(* Logix 5000 project; controller ARS14002_PLC vendor 1 type 14 code 218 rev 30.11; software revision 30.01; part 2 of 13 *)
(* tags used below, declared in another part *)
   FCV_1001 : CM_AO_VLV;
   FCV_1002 : CM_AO_VLV;
   FCV_101A : CM_AO_VLV;
   FCV_101B : CM_AO_VLV;
   FCV_101C : CM_AO_VLV;
   FCV_102A : CM_AO_VLV;
   FCV_102B : CM_AO_VLV;
   FCV_102C : CM_AO_VLV;
   FCV_1221 : CM_AO_VLV;
   FCV_1251 : CM_AO_VLV;
   FCV_202 : CM_AO_VLV;
   FCV_204 : CM_AO_VLV;
   FCV_207 : CM_AO_VLV;
   FCV_504 : CM_AO_VLV;
   FCV_603 : CM_AO_VLV;
   FCV_605 : CM_AO_VLV;
   FCV_753 : CM_AO_VLV;
   FCV_754 : CM_AO_VLV;
   FCV_755 : CM_AO_VLV;
   FT_1002 : CM_AI_SCL;
   FT_1002_MAVE : REAL;
   FT_1002_MAVE_STORAGE : REAL[30];
   FT_1221 : CM_AI_SCL;
   FT_1251 : CM_AI_SCL;
   PDT_603 : CM_AI_SCL_ALT;
   PDT_751 : CM_AI_SCL_ALT;
   PDT_753 : CM_AI_SCL_ALT;
   PT_1001 : CM_AI_SCL;
   PT_101A : CM_AI_SCL;
   PT_101B : CM_AI_SCL;
   PT_101C : CM_AI_SCL;
   PT_201 : CM_AI_SCL;
   PT_601 : CM_AI_SCL;
   PT_701 : CM_AI_SCL;
   PT_753 : CM_AI_SCL;
   PT_902 : CM_AI_SCL;
   SV_1001F : CM_DO_GENERIC;
   SV_1002F : CM_DO_GENERIC;
   SV_101AF : CM_DO_GENERIC;
   SV_101BF : CM_DO_GENERIC;
   SV_101CF : CM_DO_GENERIC;
   SV_102AF : CM_DO_GENERIC;
   SV_102BF : CM_DO_GENERIC;
   SV_102CF : CM_DO_GENERIC;
   SV_1221F : CM_DO_GENERIC;
   SV_1251F : CM_DO_GENERIC;
   SV_202F : CM_DO_GENERIC;
   SV_204F : CM_DO_GENERIC;
   SV_207F : CM_DO_GENERIC;
   SV_504F : CM_DO_GENERIC;
   SV_603F : CM_DO_GENERIC;
   SV_605F : CM_DO_GENERIC;
   SV_753F : CM_DO_GENERIC;
   SV_754F : CM_DO_GENERIC;
   SV_755F : CM_DO_GENERIC;

   TE_1250A : CM_AI_SCL := (RawMin := -4500, RawMax := 10000, EuMin := -450.0, EuMax := 1000.0, In_Raw := 487, Percent := 4.8700013, PV := 48.700012);
   TE_1250B : CM_AI_SCL := (RawMin := -4500, RawMax := 10000, EuMin := -450.0, EuMax := 1000.0, In_Raw := 520, Percent := 5.2000003, PV := 52.0);
   TE_1252 : CM_AI_SCL := (RawMin := -4500, RawMax := 10000, EuMin := -450.0, EuMax := 1000.0, In_Raw := 528, Percent := 5.279999, PV := 52.799988);
   TE_501 : CM_AI_SCL := (RawMin := -4500, RawMax := 10000, EuMin := -450.0, EuMax := 1000.0, In_Raw := 508, Percent := 5.079999, PV := 50.799988);
   TE_501_DERV : REAL := -1.000061;
   TE_501_DERV_BLOCK : DERIVATIVE := (In := 51.100006, Gain := 1.0, RTSTime := 1, Out := -1.000061, DeltaT := 0.1);
   TE_501_MAVE_BLOCK : MOVING_AVERAGE := (In := -3.000183, SampleEnable := 1, NumberOfSamples := 200, Out := 0.0049987794);
   TE_501_MAVE_STORAGE : REAL[200] := ([4] := 3.000183, [5] := 0.99975586, [8] := -0.99975586, [9] := -3.000183, [11] := 3.999939, [12] := -0.99975586, [13] := -3.000183, [14] := -1.000061, [15] := 1.000061, [16] := -1.000061, [17] := 5.0, [18] := -3.999939, [20] := 3.999939, [21] := -3.999939, [22] := 3.000183, [23] := -3.000183, [24] := 3.000183, [25] := -4.000244, [27] := 4.000244, [28] := -3.000183, [32] := 3.999939, [33] := -0.99975586, [34] := -3.000183, [36] := -1.000061, [37] := 4.000244, [39] := -3.000183, [42] := 3.000183, [45] := -3.000183, [49] := -1.000061, [50] := 1.000061, [53] := 3.999939, [55] := -3.999939, [56] := 3.000183, [60] := -3.000183, [61] := 3.000183, [63] := 0.99975586, [64] := -3.999939, [65] := 3.999939, [66] := -0.99975586, [68] := 0.99975586, [69] := -0.99975586, [70] := -3.000183, [71] := 3.000183, [75] := -3.000183, [76] := 3.000183, [77] := -3.000183, [78] := 3.000183, [79] := -3.000183, [82] := 3.000183, [84] := -4.000244, [85] := 1.000061, [89] := 3.000183, [91] := 0.99975586, [92] := -3.999939, [93] := 3.000183, [94] := -3.000183, [95] := 3.000183, [96] := -4.000244, [97] := 4.000244, [98] := -3.000183,
        [102] := 3.000183, [104] := 0.99975586, [105] := -0.99975586, [107] := -3.000183, [108] := 3.000183, [109] := -3.000183, [110] := 3.999939, [111] := -0.99975586, [114] := -4.000244, [115] := 1.000061, [116] := 3.000183, [118] := 0.99975586, [119] := -0.99975586, [122] := -3.000183, [124] := 3.000183, [125] := 0.99975586, [126] := -3.999939, [127] := 3.000183, [129] := -3.000183, [130] := 3.000183, [133] := -3.000183, [134] := 3.999939, [135] := -0.99975586, [138] := 0.99975586, [139] := -0.99975586, [141] := 0.99975586, [142] := -3.999939, [143] := 3.000183, [146] := 0.99975586, [147] := -0.99975586, [150] := -3.000183, [151] := 3.000183, [155] := 0.99975586, [158] := -0.99975586, [160] := -3.000183, [161] := 3.000183, [164] := -3.000183, [166] := 3.000183, [167] := 0.99975586, [168] := -0.99975586, [169] := -3.000183, [171] := 5.0, [172] := -5.0, [173] := -1.000061, [174] := 5.0, [175] := -0.99975586, [182] := 0.99975586, [183] := -3.999939, [185] := 3.000183, [186] := 0.99975586, [187] := -0.99975586, [189] := -3.000183, [191] := 3.000183, [193] := -3.000183, [194] := 3.999939, [195] := -3.999939, [196] := 3.000183, [197] := 0.99975586, [198] := -0.99975586);
   TE_501_MIN_SV_202 : REAL := -200.0;
   TE_501_ROC : REAL := -0.8999634;
   TE_504 : CM_AI_SCL := (RawMin := -4500, RawMax := 10000, EuMin := -450.0, EuMax := 1000.0, In_Raw := 561, Percent := 5.6100006, PV := 56.100006);
   TE_504_DERV : REAL := -3.000183;
   TE_504_DERV_BLOCK : DERIVATIVE := (In := 56.299988, Gain := 1.0, RTSTime := 1, DeltaT := 0.1);
   TE_504_MAVE_BLOCK : MOVING_AVERAGE := (SampleEnable := 1, NumberOfSamples := 1000, Out := 0.001000061, Status := 16#0000_0005, InstructFault := 1, NumberOfSampInv := 1);
   TE_504_MAVE_STORAGE : REAL[1000] := ([0] := 1.000061, [2] := -2.000122, [3] := 1.000061, [6] := 1.000061, [8] := -1.000061, [9] := -1.000061, [10] := 1.000061, [16] := 1.000061, [17] := -2.000122, [18] := 1.000061, [20] := -1.000061, [21] := 2.000122, [22] := -1.000061, [24] := -1.000061, [26] := 1.000061, [30] := 1.000061, [31] := -1.000061, [32] := -1.000061, [33] := 2.000122, [34] := -1.000061, [37] := 1.000061, [38] := -1.000061, [39] := 1.000061, [40] := -1.000061, [41] := -1.000061, [42] := 1.000061, [48] := 1.000061, [49] := -1.000061, [51] := 1.000061, [53] := -1.000061, [55] := -1.000061, [57] := 3.000183, [58] := -1.000061, [61] := -1.000061, [62] := -1.000061, [63] := 1.000061, [64] := 1.000061, [65] := -1.000061, [66] := 1.000061, [67] := -2.000122, [68] := 2.000122, [69] := -2.000122, [70] := 2.000122, [71] := -1.000061, [74] := 1.000061, [75] := -1.000061, [76] := -1.000061, [77] := 1.000061, [79] := 1.000061, [80] := -1.000061, [82] := -1.000061, [83] := 1.000061, [84] := -1.000061, [85] := 1.000061, [86] := 1.000061, [87] := -1.000061, [88] := -1.000061, [89] := 1.000061, [90] := -1.000061, [91] := 1.000061,
        [92] := 1.000061, [94] := -1.000061, [96] := 1.000061, [100] := -1.000061, [102] := 1.000061, [103] := -2.000122, [104] := 1.000061, [105] := -1.000061, [106] := 1.000061, [107] := 1.000061, [108] := -1.000061, [109] := 1.000061, [111] := -1.000061, [117] := 1.000061, [118] := -1.000061, [120] := 1.000061, [123] := -1.000061, [125] := 1.000061, [126] := -2.000122, [127] := 1.000061, [131] := 1.000061, [132] := -1.000061, [135] := 1.000061, [136] := -2.000122, [137] := 2.000122, [139] := -2.000122, [140] := 1.000061, [141] := -1.000061, [143] := 1.000061, [146] := -1.000061, [147] := 1.000061, [149] := 1.000061, [150] := -1.000061, [151] := -1.000061, [152] := 1.000061, [153] := 2.000122, [154] := -2.000122, [159] := -1.000061, [160] := 1.000061, [162] := 1.000061, [163] := -1.000061, [167] := 1.000061, [168] := -2.000122, [169] := 1.000061, [171] := 1.000061, [172] := 1.000061, [173] := -3.000183, [174] := 1.000061, [181] := -1.000061, [182] := 2.000122, [183] := -1.000061, [184] := -1.000061, [185] := 1.000061, [186] := -1.000061, [188] := 2.000122, [189] := -2.000122, [190] := 1.000061, [197] := 1.000061, [199] := -1.000061, [200] := 1.000061,
        [201] := -1.000061, [203] := 1.000061, [204] := -1.000061, [205] := 1.000061, [206] := -1.000061, [209] := 2.000122, [210] := -2.000122, [214] := -2.000122, [215] := 1.000061, [216] := 2.000122, [217] := -1.000061, [221] := 1.000061, [223] := -1.000061, [224] := 1.000061, [226] := -1.000061, [227] := -1.000061, [228] := 1.000061, [233] := 1.000061, [234] := -1.000061, [235] := 1.000061, [236] := -1.000061, [237] := 1.000061, [238] := -1.000061, [242] := -1.000061, [243] := 2.000122, [244] := -1.000061, [248] := 1.000061, [249] := -1.000061, [251] := 1.000061, [253] := -1.000061, [256] := 1.000061, [258] := 1.000061, [259] := -1.000061, [261] := -1.000061, [262] := -1.000061, [264] := 1.000061, [266] := 1.000061, [270] := -2.000122, [272] := 1.000061, [273] := 1.000061, [274] := -1.000061, [275] := -1.000061, [276] := 1.000061, [277] := 1.000061, [281] := -1.000061, [283] := -1.000061, [284] := 2.000122, [288] := -1.000061, [289] := 1.000061, [290] := -1.000061, [293] := 1.000061, [294] := -2.000122, [295] := 1.000061, [300] := 2.000122, [301] := -1.000061, [302] := -1.000061, [306] := 1.000061, [307] := -1.000061, [308] := -1.000061, [311] := 2.000122,
        [313] := -1.000061, [316] := 1.000061, [317] := -2.000122, [320] := 1.000061, [322] := -1.000061, [323] := 1.000061, [329] := 1.000061, [333] := -1.000061, [334] := 1.000061, [335] := -1.000061, [337] := 1.000061, [338] := -1.000061, [340] := 1.000061, [341] := -2.000122, [342] := 1.000061, [343] := 1.000061, [344] := -1.000061, [345] := 1.000061, [346] := -1.000061, [347] := 1.000061, [348] := -1.000061, [349] := 1.000061, [351] := -1.000061, [352] := -1.000061, [353] := 2.000122, [354] := 1.000061, [355] := -3.000183, [356] := 2.000122, [357] := -1.000061, [360] := 1.000061, [361] := -1.000061, [365] := 1.000061, [366] := -1.000061, [369] := -1.000061, [370] := 1.000061, [372] := 1.000061, [373] := -1.000061, [374] := -2.000122, [375] := 2.000122, [377] := 1.000061, [378] := -1.000061, [380] := -1.000061, [381] := 1.000061, [383] := -1.000061, [384] := 1.000061, [389] := -1.000061, [390] := 2.000122, [392] := -1.000061, [393] := 1.000061, [394] := -1.000061, [398] := -1.000061, [400] := 1.000061, [401] := -1.000061, [402] := 1.000061, [403] := 1.000061, [404] := -1.000061, [406] := 1.000061, [407] := -1.000061, [409] := -2.000122, [410] := 2.000122,
        [411] := 1.000061, [413] := -1.000061, [414] := -1.000061, [415] := 2.000122, [416] := -2.000122, [417] := 2.000122, [419] := -2.000122, [420] := 1.000061, [421] := -1.000061, [422] := 1.000061, [427] := 1.000061, [428] := -1.000061, [429] := 1.000061, [430] := -1.000061, [432] := 1.000061, [433] := -1.000061, [436] := 1.000061, [439] := -1.000061, [440] := -1.000061, [441] := 1.000061, [442] := 1.000061, [443] := -1.000061, [444] := 1.000061, [445] := -1.000061, [446] := 1.000061, [448] := -1.000061, [450] := 1.000061, [451] := -1.000061, [452] := 1.000061, [453] := -1.000061, [454] := 1.000061, [456] := -1.000061, [457] := 1.000061, [458] := -1.000061, [459] := 1.000061, [460] := -1.000061, [464] := 1.000061, [465] := 1.000061, [467] := -2.000122, [468] := 1.000061, [469] := 1.000061, [473] := -1.000061, [476] := 1.000061, [477] := -1.000061, [483] := 2.000122, [484] := -1.000061, [485] := -1.000061, [486] := 1.000061, [488] := -1.000061, [491] := 1.000061, [492] := -1.000061, [493] := -1.000061, [494] := 2.000122, [495] := -1.000061, [496] := 1.000061, [497] := -1.000061, [498] := 1.000061, [499] := -1.000061, [500] := 2.000122, [501] := -2.000122,
        [502] := 1.000061, [505] := -1.000061, [507] := 1.000061, [508] := -2.000122, [509] := 1.000061, [510] := 1.000061, [512] := -2.000122, [513] := 1.000061, [514] := 1.000061, [515] := -1.000061, [517] := -1.000061, [518] := 1.000061, [519] := 1.000061, [520] := -1.000061, [522] := -1.000061, [523] := 2.000122, [524] := -1.000061, [526] := 1.000061, [527] := -1.000061, [528] := -2.000122, [529] := 1.000061, [530] := 1.000061, [531] := 1.000061, [533] := -1.000061, [536] := -1.000061, [537] := 1.000061, [538] := 1.000061, [540] := -2.000122, [541] := 1.000061, [544] := 1.000061, [545] := -1.000061, [547] := 1.000061, [548] := -1.000061, [551] := 1.000061, [552] := -1.000061, [553] := 1.000061, [554] := -1.000061, [555] := 1.000061, [556] := -1.000061, [558] := 1.000061, [559] := -2.000122, [560] := 2.000122, [565] := -1.000061, [566] := 1.000061, [567] := -1.000061, [572] := 1.000061, [573] := -2.000122, [574] := 1.000061, [575] := 1.000061, [577] := -1.000061, [581] := 1.000061, [582] := -2.000122, [584] := 1.000061, [585] := -1.000061, [586] := 1.000061, [587] := 2.000122, [588] := -1.000061, [589] := -1.000061, [590] := 2.000122, [591] := -2.000122,
        [595] := 1.000061, [597] := -1.000061, [598] := 1.000061, [599] := -2.000122, [600] := 1.000061, [602] := -1.000061, [603] := 1.000061, [608] := -1.000061, [609] := 1.000061, [611] := 2.000122, [612] := -1.000061, [613] := -1.000061, [619] := -1.000061, [620] := 1.000061, [622] := 2.000122, [623] := -2.000122, [629] := -1.000061, [630] := 2.000122, [633] := -1.000061, [636] := 1.000061, [637] := -1.000061, [647] := -1.000061, [648] := 2.000122, [649] := -1.000061, [651] := 1.000061, [652] := -1.000061, [653] := 1.000061, [654] := -1.000061, [656] := -1.000061, [657] := 1.000061, [661] := -2.000122, [662] := 1.000061, [663] := 2.000122, [664] := -3.000183, [665] := 2.000122, [666] := 1.000061, [667] := -2.000122, [668] := 2.000122, [669] := -1.000061, [670] := -1.000061, [672] := 3.000183, [673] := -2.000122, [675] := -1.000061, [676] := 1.000061, [683] := 1.000061, [684] := -1.000061, [685] := 1.000061, [686] := -1.000061, [687] := 1.000061, [688] := -1.000061, [691] := 1.000061, [692] := -1.000061, [696] := 1.000061, [697] := -1.000061, [699] := 1.000061, [700] := -1.000061, [702] := 1.000061, [705] := -1.000061, [707] := 1.000061, [708] := -1.000061,
        [709] := 1.000061, [710] := -1.000061, [713] := 1.000061, [714] := -1.000061, [715] := 1.000061, [716] := -1.000061, [717] := -1.000061, [718] := 1.000061, [720] := 1.000061, [721] := -1.000061, [726] := 1.000061, [727] := -1.000061, [728] := -1.000061, [730] := 1.000061, [732] := 2.000122, [733] := -2.000122, [735] := 1.000061, [736] := -1.000061, [738] := -1.000061, [739] := 1.000061, [740] := 1.000061, [741] := -2.000122, [742] := 1.000061, [743] := -1.000061, [744] := 1.000061, [748] := -1.000061, [750] := 1.000061, [752] := -1.000061, [753] := 2.000122, [755] := -1.000061, [756] := -1.000061, [757] := 2.000122, [758] := -1.000061, [763] := -1.000061, [764] := 1.000061, [765] := 1.000061, [767] := -1.000061, [769] := 1.000061, [771] := -1.000061, [779] := 1.000061, [780] := -2.000122, [781] := 2.000122, [782] := -1.000061, [784] := 1.000061, [785] := -1.000061, [788] := -1.000061, [789] := 1.000061, [790] := -1.000061, [791] := 1.000061, [798] := 1.000061, [799] := -1.000061, [802] := -1.000061, [803] := 1.000061, [804] := 1.000061, [806] := -1.000061, [808] := -1.000061, [809] := 1.000061, [812] := 1.000061, [813] := -2.000122, [814] := 1.000061,
        [815] := -1.000061, [816] := 2.000122, [817] := -2.000122, [818] := 1.000061, [819] := -1.000061, [820] := 1.000061, [826] := 2.000122, [827] := -2.000122, [829] := -1.000061, [830] := 1.000061, [832] := 2.000122, [833] := -1.000061, [835] := -1.000061, [837] := 1.000061, [838] := -1.000061, [840] := 1.000061, [841] := -1.000061, [842] := 1.000061, [843] := -1.000061, [844] := -1.000061, [845] := 2.000122, [849] := -1.000061, [852] := 1.000061, [853] := -2.000122, [854] := 1.000061, [857] := -1.000061, [859] := 2.000122, [860] := -1.000061, [864] := -1.000061, [865] := 1.000061, [866] := 2.000122, [867] := -1.000061, [868] := -1.000061, [869] := 1.000061, [872] := 1.000061, [873] := -1.000061, [874] := -1.000061, [875] := 1.000061, [877] := -1.000061, [879] := 1.000061, [880] := 1.000061, [882] := -1.000061, [883] := -1.000061, [884] := 1.000061, [886] := -1.000061, [888] := 1.000061, [890] := -1.000061, [895] := -1.000061, [896] := 1.000061, [898] := -1.000061, [899] := 1.000061, [903] := -1.000061, [905] := 1.000061, [907] := -1.000061, [908] := 1.000061, [910] := 1.000061, [911] := -1.000061, [912] := -1.000061, [913] := 2.000122, [916] := 1.000061,
        [917] := -1.000061, [918] := -1.000061, [920] := 1.000061, [921] := -1.000061, [922] := -1.000061, [923] := 2.000122, [924] := -1.000061, [925] := -1.000061, [926] := 1.000061, [929] := -1.000061, [932] := 2.000122, [933] := -1.000061, [936] := 1.000061, [937] := -1.000061, [938] := -1.000061, [939] := 1.000061, [941] := -1.000061, [942] := 2.000122, [943] := -1.000061, [944] := -1.000061, [945] := 1.000061, [947] := 1.000061, [948] := -2.000122, [949] := 1.000061, [950] := 1.000061, [951] := -2.000122, [952] := 2.000122, [954] := -1.000061, [955] := 1.000061, [956] := -1.000061, [960] := -1.000061, [962] := 2.000122, [963] := -2.000122, [964] := 1.000061, [966] := 1.000061, [967] := -1.000061, [968] := 1.000061, [969] := -1.000061, [971] := -1.000061, [972] := 1.000061, [974] := 2.000122, [975] := -1.000061, [976] := -2.000122, [978] := 1.000061, [979] := -1.000061, [980] := 1.000061, [983] := 1.000061, [984] := -2.000122, [985] := 1.000061, [987] := -1.000061, [988] := 1.000061, [992] := 2.000122, [993] := -1.000061, [995] := -1.000061, [996] := -1.000061, [997] := 1.000061, [998] := 1.000061, [999] := -1.000061);
   TE_504_MAVE_STORAGE_1 : REAL[200] := ([3] := -1.000061, [4] := 1.000061, [5] := -1.000061, [6] := 2.000122, [8] := -1.000061, [10] := -1.000061, [11] := 1.000061, [20] := -1.000061, [22] := 1.000061, [27] := 1.000061, [28] := -1.000061, [29] := -1.000061, [30] := 1.000061, [32] := 1.000061, [33] := -1.000061, [34] := -1.000061, [35] := 1.000061, [36] := 1.000061, [37] := -1.000061, [40] := 1.000061, [42] := -1.000061, [44] := 1.000061, [45] := -1.000061, [50] := 1.000061, [51] := -1.000061, [52] := 1.000061, [53] := -2.000122, [56] := 1.000061, [57] := -1.000061, [58] := 1.000061, [59] := -1.000061, [61] := 1.000061, [62] := -1.000061, [64] := 2.000122, [65] := -2.000122, [66] := 1.000061, [67] := -1.000061, [68] := 1.000061, [72] := -1.000061, [73] := 1.000061, [74] := -1.000061, [76] := 1.000061, [78] := 1.000061, [79] := -1.000061, [80] := -1.000061, [82] := 1.000061, [84] := -1.000061, [85] := 1.000061, [87] := 1.000061, [88] := -1.000061, [93] := 1.000061, [94] := -1.000061, [101] := -1.000061, [102] := 1.000061, [103] := -1.000061, [104] := 1.000061, [105] := 1.000061, [106] := -2.000122, [107] := 1.000061, [108] := -1.000061,
        [109] := 1.000061, [111] := -1.000061, [113] := 1.000061, [116] := -1.000061, [117] := -1.000061, [118] := 2.000122, [119] := -1.000061, [120] := 1.000061, [122] := -1.000061, [123] := 1.000061, [125] := -1.000061, [126] := 2.000122, [128] := -1.000061, [129] := -1.000061, [130] := 1.000061, [133] := -1.000061, [134] := 1.000061, [135] := -1.000061, [139] := 1.000061, [143] := 1.000061, [144] := -1.000061, [145] := -1.000061, [146] := 1.000061, [147] := 1.000061, [148] := -2.000122, [149] := 1.000061, [152] := -1.000061, [154] := -1.000061, [155] := 2.000122, [158] := -2.000122, [159] := 2.000122, [161] := 1.000061, [163] := -1.000061, [165] := 1.000061, [166] := -1.000061, [169] := 1.000061, [170] := 1.000061, [171] := -1.000061, [175] := 2.000122, [176] := -1.000061, [178] := -1.000061, [180] := 1.000061, [183] := -1.000061, [184] := 2.000122, [185] := -2.000122, [187] := 1.000061, [188] := -2.000122, [189] := 1.000061, [191] := 1.000061, [192] := 1.000061, [193] := -2.000122, [194] := 1.000061, [195] := 1.000061, [196] := -1.000061, [197] := -1.000061, [198] := 2.000122, [199] := -1.000061);
   TE_504_ROC : REAL := 0.060003664;
   TE_601 : CM_AI_SCL := (RawMin := -4500, RawMax := 10000, EuMin := -450.0, EuMax := 1000.0, In_Raw := 732, Percent := 7.320001, PV := 73.20001);
   TE_601_DERV : REAL := -9.000244;
   TE_601_DERV_BLOCK : DERIVATIVE := (In := 74.599976, Gain := 1.0, RTSTime := 1, DeltaT := 0.1);
   TE_601_DERV_BLOCK1 : DERIVATIVE := (Gain := 1.0, RTSTime := 1);
   TE_601_DERV_BLOCK2 : DERIVATIVE := (Gain := 1.0, RTSTime := 1);
   TE_601_DERV_BLOCK3 : DERIVATIVE := (Gain := 1.0, RTSTime := 1);
   TE_601_DERV_BLOCK4 : DERIVATIVE := (Gain := 1.0, RTSTime := 1);
   TE_601_MAVE_BLOCK : MOVING_AVERAGE := (In := 5.0, SampleEnable := 1, NumberOfSamples := 200, Out := 0.005001831);
   TE_601_MAVE_STORAGE : REAL[200] := ([0] := 4.000244, [1] := -4.000244, [2] := -4.000244, [4] := -1.9995117, [5] := 8.999634, [6] := -2.999878, [9] := -7.999878, [10] := 2.999878, [11] := 10.999756, [12] := -10.999756, [13] := 7.000122, [15] := -4.000244, [16] := -2.000122, [17] := -0.99975586, [18] := 0.99975586, [19] := 6.000366, [21] := -2.999878, [22] := -3.0004883, [23] := 4.000244, [25] := -0.99975586, [26] := -2.000122, [27] := 5.999756, [28] := -5.999756, [30] := 5.0, [31] := -5.0, [32] := -1.0003662, [34] := 5.0, [35] := -2.999878, [36] := 2.000122, [37] := -2.999878, [38] := 2.000122, [39] := 1.9995117, [40] := -5.999756, [41] := 0.99975586, [42] := -2.999878, [43] := 7.999878, [44] := -5.999756, [45] := 9.000244, [46] := -1.0003662, [47] := -0.99975586, [48] := -2.000122, [49] := 2.000122, [50] := -7.000122, [51] := 2.999878, [52] := 2.999878, [53] := 1.0003662, [54] := -4.000244, [56] := -2.000122, [57] := 3.0004883, [58] := 0.99975586, [59] := -2.999878, [60] := 5.0, [61] := -6.000366, [62] := 6.000366, [63] := -5.0, [64] := 7.000122, [65] := -8.000488, [66] := 7.000122, [67] := -5.0, [68] := 1.0003662,
        [69] := 1.9995117, [71] := -2.999878, [72] := 1.0003662, [73] := 0.99975586, [74] := -0.99975586, [75] := -1.0003662, [76] := -0.99975586, [77] := 2.000122, [78] := -1.0003662, [79] := 5.0, [80] := -5.0, [81] := -0.99975586, [82] := 0.99975586, [84] := -0.99975586, [86] := 7.000122, [87] := -3.0004883, [89] := -1.9995117, [90] := 2.999878, [91] := -5.0, [92] := 3.9996338, [93] := -3.9996338, [94] := 2.000122, [95] := -2.000122, [96] := -1.0003662, [97] := 1.0003662, [98] := 0.99975586, [99] := 2.000122, [100] := -0.99975586, [101] := -3.0004883, [102] := 11.000366, [103] := 5.999756, [104] := -5.999756, [105] := 3.9996338, [106] := -0.99975586, [107] := -2.000122, [108] := -0.99975586, [109] := 2.999878, [110] := -1.0003662, [111] := -0.99975586, [114] := 0.99975586, [115] := -1.9995117, [116] := 10.0, [117] := -6.000366, [119] := -3.9996338, [120] := 7.999878, [121] := -1.0003662, [122] := 5.0, [123] := -3.9996338, [124] := -7.000122, [125] := 0.99975586, [126] := -0.99975586, [128] := 7.999878, [129] := -10.0, [130] := 10.0, [131] := -7.000122, [132] := -2.999878, [133] := 9.000244, [134] := -7.000122, [135] := 7.999878, [136] := -2.999878,
        [137] := -5.999756, [138] := 1.9995117, [139] := -0.99975586, [140] := 7.999878, [141] := 1.0003662, [143] := -4.000244, [144] := -2.000122, [145] := -5.0, [146] := 2.999878, [147] := 3.0004883, [148] := -5.0, [149] := 2.999878, [150] := 5.0, [151] := -2.999878, [152] := 0.99975586, [153] := -2.000122, [154] := 1.0003662, [155] := -3.0004883, [156] := 1.0003662, [157] := 5.999756, [158] := -12.999878, [159] := 7.999878, [160] := -3.9996338, [161] := 12.999878, [162] := -5.0, [163] := -6.000366, [164] := -0.99975586, [165] := 2.999878, [166] := -2.999878, [167] := 7.000122, [168] := -2.999878, [169] := -2.000122, [170] := 2.999878, [171] := -5.0, [172] := 4.000244, [173] := 2.999878, [175] := -2.999878, [176] := 3.9996338, [177] := -7.999878, [178] := 7.000122, [179] := 2.000122, [180] := -8.000488, [184] := 2.000122, [187] := -0.99975586, [189] := 5.0, [190] := -6.000366, [191] := 7.000122, [192] := -7.000122, [193] := -0.99975586, [194] := 0.99975586, [195] := 1.0003662, [196] := -2.000122, [199] := 5.0);
   TE_601_ROC : REAL := 2.0998533;
   TE_602 : CM_AI_SCL := (RawMin := -4500, RawMax := 10000, EuMin := -450.0, EuMax := 1000.0, In_Raw := -2046, Percent := -20.460001, PV := -204.6);
   TE_602_DERV : REAL;
   TE_602_DERV_BLOCK : DERIVATIVE := (In := -198.4, Gain := 1.0, RTSTime := 1, Out := -0.99990845, DeltaT := 0.1);
   TE_602_MAVE_BLOCK : MOVING_AVERAGE := (SampleEnable := 1, NumberOfSamples := 200, Out := 0.0800003);
   TE_602_MAVE_STORAGE : REAL[200] := ([0] := -2.000122, [1] := 4.0000916, [3] := -4.0000916, [5] := 2.000122, [7] := -2.000122, [9] := 2.000122, [10] := -2.000122, [11] := 4.0000916, [12] := -1.9999695, [16] := 1.9999695, [17] := -4.0000916, [18] := 2.000122, [21] := 1.9999695, [22] := -1.9999695, [23] := 1.9999695, [24] := -1.9999695, [25] := 1.9999695, [26] := -1.9999695, [27] := -1.9999695, [28] := 3.999939, [29] := -1.9999695, [30] := 1.9999695, [31] := -3.999939, [32] := 1.9999695, [34] := -1.9999695, [35] := 3.999939, [36] := -1.9999695, [40] := -3.999939, [41] := 5.9999084, [42] := -1.9999695, [45] := 1.9999695, [46] := -3.999939, [47] := 1.9999695, [50] := 1.9999695, [53] := -1.9999695, [54] := 1.9999695, [55] := -1.9999695, [57] := 1.9999695, [62] := -1.9999695, [63] := 3.999939, [65] := -1.9999695, [67] := 1.9999695, [68] := -1.9999695, [69] := 1.9999695, [70] := -3.999939, [71] := 3.999939, [75] := -1.9999695, [78] := 1.9999695, [81] := -1.9999695, [83] := -1.9999695, [84] := 3.999939, [85] := -1.9999695, [87] := 1.9999695, [91] := -1.9999695, [92] := 1.9999695, [97] := 1.000061, [98] := -1.000061, [99] := 1.000061, [102] := -1.000061, [104] := 1.000061,
        [105] := -1.000061, [107] := 1.000061, [108] := -1.000061, [110] := 3.0000305, [112] := -5.0, [113] := 3.0000305, [115] := 1.9999695, [116] := -1.9999695, [117] := -1.000061, [118] := 1.000061, [120] := -3.0000305, [121] := 5.0, [123] := -1.9999695, [124] := 1.9999695, [125] := -1.9999695, [126] := -1.000061, [127] := -1.9999695, [128] := 3.0000305, [129] := -1.000061, [130] := 1.000061, [131] := -1.000061, [132] := 1.000061, [133] := 1.9999695, [134] := -1.9999695, [137] := 3.999939, [138] := -1.9999695, [139] := 1.9999695, [140] := -3.999939, [144] := 1.9999695, [145] := -1.9999695, [147] := 1.9999695, [148] := -1.9999695, [149] := 1.9999695, [150] := -1.9999695, [151] := 1.9999695, [152] := 1.9999695, [153] := -1.9999695, [156] := -1.9999695, [158] := 1.9999695, [159] := 4.0000916, [160] := -2.000122, [161] := -1.9999695, [166] := 1.9999695, [167] := -1.9999695, [169] := -1.9999695, [170] := 3.999939, [172] := -1.9999695, [173] := 1.9999695, [175] := 2.000122, [176] := -2.000122, [177] := -1.9999695, [183] := 4.0000916, [184] := -2.000122, [185] := -1.9999695, [187] := 1.9999695, [190] := 2.000122, [191] := -2.000122, [192] := 4.0000916, [193] := -4.0000916, [196] := -1.9999695,
        [197] := 1.9999695, [199] := 2.000122);
   TE_602_ROC : REAL := 2.6999815;
   TE_604 : CM_AI_SCL := (RawMin := -4500, RawMax := 10000, EuMin := -450.0, EuMax := 1000.0, In_Raw := 732, Percent := 7.320001, PV := 73.20001);
   TE_604_DERV : REAL := 1.0003662;
   TE_604_DERV_BLOCK : DERIVATIVE := (In := 73.29999, Gain := 1.0, RTSTime := 1, DeltaT := 0.1);
   TE_604_MAVE_BLOCK : MOVING_AVERAGE := (In := -2.000122, SampleEnable := 1, NumberOfSamples := 200, Out := -0.0049987794);
   TE_604_MAVE_STORAGE : REAL[200] := ([1] := -2.000122, [2] := 2.000122, [6] := -1.0003662, [9] := 2.000122, [11] := -2.000122, [12] := -2.000122, [13] := 2.000122, [15] := 1.0003662, [16] := -1.0003662, [17] := 1.0003662, [20] := 0.99975586, [21] := -2.000122, [23] := 1.0003662, [28] := -1.0003662, [32] := 1.0003662, [34] := -1.0003662, [35] := 1.0003662, [36] := -2.000122, [37] := 0.99975586, [39] := 1.0003662, [40] := -1.0003662, [42] := 1.0003662, [43] := -2.000122, [45] := 2.999878, [46] := -2.000122, [49] := 1.0003662, [50] := -1.0003662, [51] := 1.0003662, [52] := -2.000122, [53] := 0.99975586, [55] := 1.0003662, [57] := 0.99975586, [58] := -0.99975586, [59] := -2.000122, [60] := 0.99975586, [61] := 1.0003662, [62] := 0.99975586, [63] := -2.000122, [66] := 1.0003662, [67] := -2.000122, [68] := 2.000122, [70] := -1.0003662, [73] := 2.000122, [76] := -2.000122, [77] := -0.99975586, [78] := 2.000122, [79] := 0.99975586, [80] := -2.000122, [81] := -0.99975586, [83] := 2.999878, [84] := -0.99975586, [85] := -1.0003662, [86] := -2.000122, [87] := 2.000122, [88] := 1.0003662, [89] := -1.0003662, [93] := -0.99975586, [94] := 0.99975586, [95] := -0.99975586, [96] := 2.000122,
        [97] := -2.000122, [101] := 0.99975586, [103] := -0.99975586, [104] := 2.000122, [105] := -1.0003662, [107] := 1.0003662, [109] := -2.000122, [110] := 0.99975586, [111] := -2.999878, [112] := 2.000122, [114] := -1.0003662, [115] := 2.000122, [116] := -0.99975586, [117] := -1.0003662, [118] := -2.000122, [119] := 3.0004883, [120] := -1.0003662, [121] := 1.0003662, [123] := -2.000122, [124] := 2.000122, [125] := 0.99975586, [126] := -0.99975586, [127] := 0.99975586, [128] := -2.000122, [129] := -0.99975586, [130] := 0.99975586, [131] := 2.999878, [133] := -2.999878, [136] := 1.0003662, [137] := -2.000122, [138] := 0.99975586, [142] := 1.0003662, [144] := 0.99975586, [145] := -0.99975586, [146] := -1.0003662, [151] := 1.0003662, [152] := -1.0003662, [155] := 1.0003662, [156] := -2.000122, [157] := 0.99975586, [158] := 1.0003662, [162] := -1.0003662, [163] := 1.0003662, [164] := -1.0003662, [167] := 1.0003662, [168] := -3.0004883, [169] := 2.000122, [170] := 1.0003662, [171] := -2.000122, [173] := 0.99975586, [174] := -0.99975586, [175] := 2.000122, [176] := -2.000122, [177] := 0.99975586, [178] := -0.99975586, [179] := 2.000122, [181] := -2.000122, [182] := 0.99975586, [185] := 1.0003662, [187] := -1.0003662,
        [188] := -0.99975586, [189] := 2.000122, [192] := -2.000122, [193] := 2.999878, [194] := -2.999878, [196] := 2.000122, [198] := -1.0003662, [199] := 1.0003662);
   TE_604_ROC : REAL;
   TE_609 : CM_AI_SCL := (RawMin := -4500, RawMax := 10000, EuMin := -450.0, EuMax := 1000.0, In_Raw := 440, Percent := 4.4, PV := 44.0);
   TE_801A : CM_AI_SCL := (RawMin := -4500, RawMax := 10000, EuMin := -450.0, EuMax := 1000.0, In_Raw := 507, Percent := 5.070001, PV := 50.700012);
   TE_801B : CM_AI_SCL := (RawMin := -4500, RawMax := 10000, EuMin := -450.0, EuMax := 1000.0, In_Raw := 508, Percent := 5.079999, PV := 50.799988);
   TE_801C : CM_AI_SCL := (RawMin := -4500, RawMax := 10000, EuMin := -450.0, EuMax := 1000.0, In_Raw := 517, Percent := 5.170001, PV := 51.700012);
   TE_801D : CM_AI_SCL := (RawMin := -4500, RawMax := 10000, EuMin := -450.0, EuMax := 1000.0, In_Raw := 522, Percent := 5.220001, PV := 52.200012);
   TE_802_INIT_TEMP : REAL := -80.0;
   TE_802A : CM_AI_SCL := (RawMin := -4500, RawMax := 10000, EuMin := -450.0, EuMax := 1000.0, In_Raw := 509, Percent := 5.089999, PV := 50.899994);
   TE_802B : CM_AI_SCL := (RawMin := -4500, RawMax := 10000, EuMin := -450.0, EuMax := 1000.0, In_Raw := 515, Percent := 5.15, PV := 51.5);
   TE_802C : CM_AI_SCL := (RawMin := -4500, RawMax := 10000, EuMin := -450.0, EuMax := 1000.0, In_Raw := 506, Percent := 5.060001, PV := 50.600006);
   TE_802D : CM_AI_SCL := (RawMin := -4500, RawMax := 10000, EuMin := -450.0, EuMax := 1000.0, In_Raw := 517, Percent := 5.170001, PV := 51.700012);
   TE_803_XV_721A_BURP_SP : REAL := -260.0;
   TE_803A : CM_AI_SCL := (RawMin := -4500, RawMax := 10000, EuMin := -450.0, EuMax := 1000.0, In_Raw := 515, Percent := 5.15, PV := 51.5);
   TE_803B : CM_AI_SCL := (RawMin := -4500, RawMax := 10000, EuMin := -450.0, EuMax := 1000.0, In_Raw := 538, Percent := 5.3799987, PV := 53.799988);
   TE_803C : CM_AI_SCL := (RawMin := -4500, RawMax := 10000, EuMin := -450.0, EuMax := 1000.0, In_Raw := 526, Percent := 5.2600007, PV := 52.600006);
   TE_803D : CM_AI_SCL := (RawMin := -4500, RawMax := 10000, EuMin := -450.0, EuMax := 1000.0, In_Raw := 543, Percent := 5.429999, PV := 54.299988);
   TE_804_INIT_TEMP : REAL := -80.0;
   TE_804A : CM_AI_SCL := (RawMin := -4500, RawMax := 10000, EuMin := -450.0, EuMax := 1000.0, In_Raw := 520, Percent := 5.2000003, PV := 52.0);
   TE_804B : CM_AI_SCL := (RawMin := -4500, RawMax := 10000, EuMin := -450.0, EuMax := 1000.0, In_Raw := 518, Percent := 5.179999, PV := 51.799988);
   TE_804C : CM_AI_SCL := (RawMin := -4500, RawMax := 10000, EuMin := -450.0, EuMax := 1000.0, In_Raw := 522, Percent := 5.220001, PV := 52.200012);
   TE_804D : CM_AI_SCL := (RawMin := -4500, RawMax := 10000, EuMin := -450.0, EuMax := 1000.0, In_Raw := 528, Percent := 5.279999, PV := 52.799988);
   TE_901 : CM_AI_SCL := (RawMin := -4500, RawMax := 10000, EuMin := -450.0, EuMax := 1000.0, In_Raw := 576, Percent := 5.7600007, PV := 57.600006);
   TE_901_InRange : BOOL;
   TE_901_SPH : REAL := -180.0;
   TE_901_SPL : REAL := -194.0;
   TE_902 : CM_AI_SCL := (RawMin := -4500, RawMax := 10000, EuMin := -450.0, EuMax := 1000.0, In_Raw := 560, Percent := 5.6000004, PV := 56.0);
   TE_903 : CM_AI_SCL := (RawMin := -4500, RawMax := 10000, EuMin := -450.0, EuMax := 1000.0, In_Raw := 558, Percent := 5.5799985, PV := 55.799988);
   TE_904 : CM_AI_SCL := (RawMin := -4500, RawMax := 10000, EuMin := -450.0, EuMax := 1000.0, In_Raw := 585, Percent := 5.85, PV := 58.5);
   TE_T_Fail_Temp : DINT := 700;
   TE_T_RAWMAX : INT := 10000;
   TE_T_RAWMIN : INT := -4500;
   TEST_COOLDOWN_ALT : BOOL;
   TEST_DERV_BLOCK : DERIVATIVE := (In := 2863.5427, Gain := 1.0, RTSTime := 1, Out := 1.0009766, DeltaT := 0.1);
   TEST_DERV_IN : REAL := 2863.6428;
   TEST_DERV_OUT : REAL := 1.0009766;
   TIME_TO_GOOD_GAS_AT2 : REAL := 10000.0;
   TIME_TO_GOOD_GAS_AT3 : REAL := 10000.0;
   TIME_TO_GOOD_GAS_PILOT : REAL := 10000.0;
   TimeStamp : DINT[7] := ([0] := 2020, [1] := 5, [2] := 1, [3] := 15, [4] := 43, [5] := 17, [6] := 945571);
   TK_1000_SCF : REAL := 47616.055;   // TOTAL SCF IN BUFFER
   TK_1100A_Low : BOOL;
   TK_1100A_LOW_DLA_TMR : TIMER := (PRE := 15000);
   TK_1100A_Low_SPH : REAL := 40.0;
   TK_1100A_Low_SPL : REAL := 30.0;
   TK_1100A_Low_Warning : BOOL;
   TK_1100A_LOW_WARNING_DLA_TMR : TIMER := (PRE := 15000);
   TK_1100A_Low_WARNING_SPH : REAL := 80.0;
   TK_1100A_Low_WARNING_SPL : REAL := 70.0;
   TK_1100A_PBC_Pressure_SPH : INT := 30;
   TK_1100A_PBC_Pressure_SPL : INT := 25;
   TK_1100A_Vent_Closed_TMR : TIMER := (PRE := 10000, ACC := 10000, EN := 1, DN := 1);
   TK_1100A_Vent_Open_TMR : TIMER := (PRE := 10000);
   TK_1100A_Vent_Pressure_SPH : INT := 50;
   TK_1100A_Vent_Pressure_SPL : INT := 45;
   TK_1300A_PBC_Pressure_SPH : INT := 42;
   TK_1300A_PBC_Pressure_SPL : INT := 40;
   TK_1300A_Vent_Closed_TMR : TIMER := (PRE := 10000, ACC := 10000, EN := 1, DN := 1);
   TK_1300A_Vent_Open_TMR : TIMER := (PRE := 10000);
   TK_1300A_Vent_Pressure_SPH : INT := 48;
   TK_1300A_Vent_Pressure_SPL : INT := 46;
   TK_1300B_Vent_Closed_TMR : TIMER := (PRE := 10000, ACC := 10000, EN := 1, DN := 1);
   TK_1300B_Vent_Open_TMR : TIMER := (PRE := 10000);
   TK_220_FILLS_MONTH : COUNTER := (PRE := 100000, ACC := 271);
   TK_220_Pressure_SPH : INT := 80;
   TK_220_Pressure_SPL : INT := 55;
   TK_700_AUTOFILL : BOOL;   // 1= TK-1100A WILL FILL TK-700
   TK_700_AUTOFILL_PDT_601_ALT_SPH : REAL := 150.0;
   TK_700_AUTOFILL_SPH : REAL := 500.0;
   TK_700_AUTOFILL_SPL : REAL := 400.0;
   TK_700_AUTOSOURCE_SPH : REAL := 1000.0;   // Level where source will switch back to TK-700
   TK_700_AUTOSOURCE_SPL : REAL := 350.0;   // Level where source will switch away from TK-700
   TK_700_FILLREQ : BOOL;
   TK_700_Full : BOOL;
   TK_700_FULL_DLA_TMR : TIMER := (PRE := 15000);
   TK_700_Full_SPH : REAL := 200.0;
   TK_700_Full_SPL : REAL := 195.0;
   TK_700_Low : BOOL := 1;
   TK_700_LOW_DLA_TMR : TIMER := (PRE := 15000, ACC := 15000, EN := 1, DN := 1);
   TK_700_Low_SPH : REAL := 35.0;
   TK_700_Low_SPL : REAL := 20.0;
   TK_700_NOT_FULL_DLA_TMR : TIMER := (PRE := 15000, ACC := 15000, EN := 1, DN := 1);
   TK_700_OVERFULL_DLA_TMR : TIMER := (PRE := 15000);
   TK_700_RETURN_SPH : REAL := 1050.0;
   TK_700_RETURN_SPH_SUB : REAL := 900.0;
   TK_700_RETURN_SPL : REAL := 500.0;
   TK_700_RETURN_SPL_PLUS : REAL := 550.0;
   VAPORIZER_WATER_DIFFERENTIAL : REAL := -2.600006;
   VENT_COLLECTION_CERTAIN_SP : REAL := 5.0;
   VENT_COLLECTION_LIKELY_SP : REAL := 15.0;
   VFD800A_ChangeDir : BOOL;
   VFD800A_ChangeDirOnStop : BOOL;
   VFD800A_ClearFault_Reset_TMR : TIMER := (PRE := 5000);
   VFD800A_CommFlt_TON : TIMER := (PRE := 10000);
   VFD800A_COMMLOSS : BOOL;
   VFD800A_DCBusVolts_HoldingRegister : DINT := 677;
   VFD800A_RunTime_CalcHigh : DINT := 3500;
   VFD800A_RunTime_CalcLow : DINT := 3400;
   VFD800A_RunTime_Modulo : DINT;
   VFD800A_RunTime_x100Hrs_Current : DINT := 33;
   VFD800A_RunTime_x100Hrs_Last : DINT;
   VFD800A_RunTime_x100Hrs_PlusOne : DINT;
   VFD800B_ChangeDir : BOOL;
   VFD800B_ChangeDirOnStop : BOOL;
   VFD800B_ClearFault_Reset_TMR : TIMER := (PRE := 5000);
   VFD800B_CommFlt_TON : TIMER := (PRE := 10000);
   VFD800B_COMMLOSS : BOOL;
   VFD800B_DCBusVolts_HoldingRegister : DINT := 677;
   VFD800B_RunTime_CalcHigh : DINT := 1200;
   VFD800B_RunTime_CalcLow : DINT := 1100;
   VFD800B_RunTime_Modulo : DINT;
   VFD800B_RunTime_x100Hrs_Current : DINT := 10;
   VFD800B_RunTime_x500Hrs_Last : DINT;
   VFD_800A_Auto : BOOL := 1;
   VFD_800A_Auto_ONS : BOOL;
   VFD_800A_AutoReq : BOOL;
   VFD_800A_ClearFault_TMR : TIMER := (PRE := 60000);
   VFD_800A_COMMLOSS : BOOL;
   VFD_800A_DISABLE_ONS : BOOL := 1;
   VFD_800A_EN : BOOL;
   VFD_800A_ManReq : BOOL;
   VFD_800A_ManStartReq : BOOL;
   VFD_800A_ST : BOOL;
   VFD_800B_Auto : BOOL;
   VFD_800B_Auto_ONS : BOOL := 1;
   VFD_800b_AutoReq : BOOL;
   VFD_800B_ClearFault_TMR : TIMER := (PRE := 60000);
   VFD_800B_COMMLOSS : BOOL;
   VFD_800B_DISABLE_ONS : BOOL := 1;
   VFD_800B_EN : BOOL;
   VFD_800B_ManReq : BOOL;
   VFD_800B_ManStartReq : BOOL;
   VFD_800B_ST : BOOL;
   WATCHDOG_1000_TON1 : TIMER := (PRE := 7500, ACC := 445, EN := 1, TT := 1);
   WATCHDOG_1000_TON2 : TIMER := (PRE := 7500);
   WATCHDOG_100_TON1 : TIMER := (PRE := 7500, ACC := 1913, EN := 1, TT := 1);
   WATCHDOG_100_TON2 : TIMER := (PRE := 7500);
   WATCHDOG_600_TON1 : TIMER := (PRE := 7500, ACC := 1843, EN := 1, TT := 1);
   WATCHDOG_600_TON2 : TIMER := (PRE := 7500);
   WATCHDOG_800_TON1 : TIMER := (PRE := 7500);
   WATCHDOG_800_TON2 : TIMER := (PRE := 7500);
   WATCHDOG_AT2_TO_ARS_OUT : BOOL;
   WATCHDOG_AT2_TO_ARS_TON1 : TIMER := (PRE := 7500);
   WATCHDOG_AT2_TO_ARS_TON2 : TIMER := (PRE := 7500);
   WATCHDOG_AT3_TO_ARS_OUT : BOOL;
   WATCHDOG_AT3_TO_ARS_TON1 : TIMER := (PRE := 7500);
   WATCHDOG_AT3_TO_ARS_TON2 : TIMER := (PRE := 7500);
   WATCHDOG_FROM_ARS_IN : BOOL;
   WATCHDOG_IN_100 : BOOL;
   WATCHDOG_IN_1000 : BOOL;
   WATCHDOG_IN_600 : BOOL;
   WATCHDOG_IN_800 : BOOL;
   WATCHDOG_OUT_100 : BOOL;
   WATCHDOG_OUT_1000 : BOOL;
   WATCHDOG_OUT_600 : BOOL;
   WATCHDOG_OUT_800 : BOOL;
   WATCHDOG_OUT_HMI : BOOL;
   WATCHDOG_OUT_MCP : BOOL;
   WATCHDOG_PILOT_TO_ARS_OUT : BOOL;
   WATCHDOG_PILOT_TO_ARS_TON1 : TIMER := (PRE := 7500);
   WATCHDOG_PILOT_TO_ARS_TON2 : TIMER := (PRE := 7500);
   WATCHDOG_TOF : TIMER := (PRE := 2500, ACC := 2500);
   WATCHDOG_TON : TIMER := (PRE := 2500, ACC := 1595, EN := 1, TT := 1);
   XV_1001 : CM_DO_VLV := (Auto := 1, Open := 1, Closed := 1, AlmCD_TmrPre := 5, EnergizeReq := 1, AlmCD := 1, Out := 1);
   XV_101B : CM_DO_VLV := (FailPos := 1, AlmCD_TmrPre := 20, EnergizeReq := 1, AlmCD := 1);
   XV_101C : CM_DO_VLV := (FailPos := 1, AlmCD_TmrPre := 20, EnergizeReq := 1, AlmCD := 1);
   XV_1123 : CM_DO_VLV := (Auto := 1, Open := 1, AlmCD_TmrPre := 5, EnergizeReq := 1, Out := 1);
   XV_1201 : CM_DO_VLV := (Open := 1, AlmCD_TmrPre := 5, Out := 1);
   XV_1202 : CM_DO_VLV := (Closed := 1, AlmCD_TmrPre := 5);
   XV_1203 : CM_DO_VLV := (Closed := 1, AlmCD_TmrPre := 5, EnergizeReq := 1);
   XV_1204 : CM_DO_VLV := (Closed := 1, AlmCD_TmrPre := 5);
   XV_1205 : CM_DO_VLV := (Closed := 1, AlmCD_TmrPre := 5);
   XV_505_PT_603_SPH_VENT : REAL := 70.0;
   XV_505_PT_603_SPL_VENT : REAL := 65.0;
   XV_623 : CM_DO_VLV := (Auto := 1, Closed := 1, AlmCD_TmrPre := 5);
   XV_623_FILL_MODE : BOOL;   // (0=Manual, 1=Auto)
   XV_623_SPH : INT := 30;
   XV_623_SPL : INT := 2;
   XV_703 : CM_DO_VLV := (Open := 1, AlmCD_TmrPre := 5, Out := 1);
   XV_721_BURP_AUTO : BOOL := 1;
   XV_721A : CM_DO_VLV := (Auto := 1, Closed := 1, AlmCD_TmrPre := 5);
   XV_721B : CM_DO_VLV := (Closed := 1, AlmCD_TmrPre := 5, EnergizeReq := 1);
   XV_801A : CM_DO_VLV := (Auto := 1, Closed := 1, AlmCD_TmrPre := 5);
   XV_801B : CM_DO_VLV := (Auto := 1, Closed := 1, AlmCD_TmrPre := 5);
   XV_801C : CM_DO_VLV := (Auto := 1, Closed := 1, AlmCD_TmrPre := 5);
   XV_801D : CM_DO_VLV := (Auto := 1, AlmCD_TmrPre := 5, AlmCD := 1);
   XV_802_VENT_COUNTER : COUNTER := (PRE := 1000000, ACC := 10903);
   XV_802_VENT_TOTAL_TIME : TIMER := (PRE := 1000000000, ACC := 1000000000, DN := 1);
   XV_806 : CM_DO_VLV := (Auto := 1, Closed := 1, AlmCD_TmrPre := 5);
   XV_806_SPH_802_CLOSED : REAL := 150.0;
   XV_806_SPH_802_OPEN : REAL := 135.0;
   XV_806_SPL_802_CLOSED : REAL := 135.0;
   XV_806_SPL_802_OPEN : REAL := 120.0;
   ZT_1001 : CM_AI_SCL := (RawMin := 4000, RawMax := 20000, EuMax := 100.0, In_Raw := 19816, Percent := 98.85, PV := 98.85);
   ZT_1002 : CM_AI_SCL := (RawMin := 4000, RawMax := 20000, EuMax := 100.0, In_Raw := 9635, Percent := 35.21875, PV := 35.21875);
   ZT_101A : CM_AI_SCL := (RawMin := 4000, RawMax := 20000, EuMax := 100.0, In_Raw := 3995, Percent := -0.03125, PV := -0.03125);
   ZT_101B : CM_AI_SCL := (RawMin := 4000, RawMax := 20000, EuMax := 100.0, In_Raw := 4844, Percent := 5.275, PV := 5.275);
   ZT_101C : CM_AI_SCL := (RawMin := 4000, RawMax := 20000, EuMax := 100.0, In_Raw := 4199, Percent := 1.24375, PV := 1.24375);
   ZT_102A : CM_AI_SCL := (RawMin := 4000, RawMax := 20000, EuMax := 100.0, In_Raw := 3997, Percent := -0.01875, PV := -0.01875);
   ZT_102B : CM_AI_SCL := (RawMin := 4000, RawMax := 20000, EuMax := 100.0, In_Raw := 3738, Percent := -1.6374999, PV := -1.6375);
   ZT_102C : CM_AI_SCL := (RawMin := 4000, RawMax := 20000, EuMax := 100.0, In_Raw := 3969, Percent := -0.19375, PV := -0.19375);
   ZT_1221 : CM_AI_SCL := (RawMin := 4000, RawMax := 20000, EuMax := 100.0, In_Raw := 3793, Percent := -1.29375, PV := -1.29375);
   ZT_1251 : CM_AI_SCL := (RawMin := 4000, RawMax := 20000, EuMax := 100.0, In_Raw := 4333, Percent := 2.08125, PV := 2.08125);
   ZT_202 : CM_AI_SCL := (RawMin := 4000, RawMax := 20000, EuMax := 100.0, In_Raw := 3992, Percent := -0.05, PV := -0.05);
   ZT_204 : CM_AI_SCL := (RawMin := 4000, RawMax := 20000, EuMax := 100.0, In_Raw := 4069, Percent := 0.43124998, PV := 0.43125);
   ZT_207 : CM_AI_SCL := (RawMin := 4000, RawMax := 20000, EuMax := 100.0, In_Raw := 4083, Percent := 0.51875, PV := 0.51875);
   ZT_504 : CM_AI_SCL := (RawMin := 4000, RawMax := 20000, EuMax := 100.0, In_Raw := 5602, Percent := 10.0125, PV := 10.0125);
   ZT_603 : CM_AI_SCL := (RawMin := 4000, RawMax := 20000, EuMax := 100.0, In_Raw := 13419, Percent := 58.868755, PV := 58.86875);
   ZT_605 : CM_AI_SCL := (RawMin := 4000, RawMax := 20000, EuMax := 100.0, In_Raw := 3994, Percent := -0.0375, PV := -0.0375);
   ZT_753 : CM_AI_SCL := (RawMin := 4000, RawMax := 20000, EuMax := 100.0, In_Raw := 3998, Percent := -0.0125, PV := -0.0125);
   ZT_754 : CM_AI_SCL := (RawMin := 4000, RawMax := 20000, EuMax := 100.0, In_Raw := 3735, Percent := -1.6562499, PV := -1.65625);
   ZT_755 : CM_AI_SCL := (RawMin := 4000, RawMax := 20000, EuMax := 100.0, In_Raw := 4553, Percent := 3.4562497, PV := 3.45625);
END_VAR

PROGRAM MainProgPeriodic   (* main routine MainRoutinePeriodic *)
VAR
   ADD_01 : FBD_MATH := (SourceA := 125.03422, SourceB := 1.0, Dest := 126.03422);
   ADD_02 : FBD_MATH := (SourceA := 0.1, SourceB := 2863.5427, Dest := 2863.6428);
   DERV_01 : DERIVATIVE := (Gain := 1.0, RTSTime := 1);
   DERV_02 : DERIVATIVE := (Gain := 1.0, RTSTime := 1);
   MAVE_01 : MOVING_AVERAGE := (SampleEnable := 1, NumberOfSamples := 1);
   MAVE_02 : MOVING_AVERAGE := (SampleEnable := 1, NumberOfSamples := 1);
   MAVE_03 : MOVING_AVERAGE := (SampleEnable := 1, NumberOfSamples := 1);
   MAVE_04 : MOVING_AVERAGE := (SampleEnable := 1, NumberOfSamples := 1);
   MAVE_05 : MOVING_AVERAGE := (SampleEnable := 1, NumberOfSamples := 1);
   MAVE_06 : MOVING_AVERAGE := (SampleEnable := 1, NumberOfSamples := 1);
   MUL_01 : FBD_MATH := (SourceA := 0.015000915, SourceB := 60.0, Dest := 0.90005493);
   MUL_02 : FBD_MATH := (SourceA := 0.001000061, SourceB := 60.0, Dest := 0.060003664);
   MUL_03 : FBD_MATH := (SourceB := 60.0);
   MUL_04 : FBD_MATH := (SourceA := 0.05499954, SourceB := 60.0, Dest := 3.2999725);
   MUL_05 : FBD_MATH := (SourceA := -0.019998169, SourceB := 60.0, Dest := -1.1998901);
   MUL_06 : FBD_MATH := (SourceA := -0.0049591064, SourceB := 60.0, Dest := -0.2975464);
   MUL_07 : FBD_MATH := (SourceA := 0.0049591064, SourceB := 60.0, Dest := 0.2975464);
   MUL_08 : FBD_MATH := (SourceA := 0.03501892, SourceB := 60.0, Dest := 2.1011353);
   MUL_09 : FBD_MATH := (SourceA := -0.0049972534, SourceB := 60.0, Dest := -0.2998352);
   MUL_10 : FBD_MATH := (SourceA := 0.0049972534, SourceB := 60.0, Dest := 0.2998352);
END_VAR

ROUTINE _13_Inputs_Mov_Avg   (* function block diagram *)
   SHEET 1
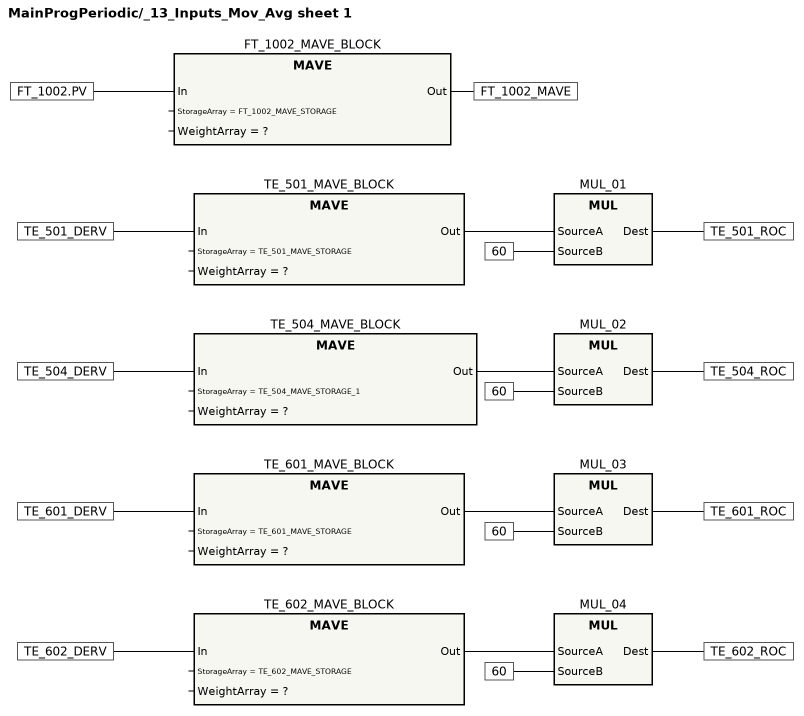
   FT_1002_MAVE_BLOCK : MAVE(In := FT_1002.PV, StorageArray := FT_1002_MAVE_STORAGE, WeightArray := ?);
   TE_501_MAVE_BLOCK : MAVE(In := TE_501_DERV, StorageArray := TE_501_MAVE_STORAGE, WeightArray := ?);
   TE_504_MAVE_BLOCK : MAVE(In := TE_504_DERV, StorageArray := TE_504_MAVE_STORAGE_1, WeightArray := ?);
   TE_601_MAVE_BLOCK : MAVE(In := TE_601_DERV, StorageArray := TE_601_MAVE_STORAGE, WeightArray := ?);
   TE_602_MAVE_BLOCK : MAVE(In := TE_602_DERV, StorageArray := TE_602_MAVE_STORAGE, WeightArray := ?);
   FT_1002_MAVE := FT_1002_MAVE_BLOCK.Out;
   MUL_01 : MUL(SourceA := TE_501_MAVE_BLOCK.Out, SourceB := 60);
   MUL_02 : MUL(SourceA := TE_504_MAVE_BLOCK.Out, SourceB := 60);
   MUL_03 : MUL(SourceA := TE_601_MAVE_BLOCK.Out, SourceB := 60);
   MUL_04 : MUL(SourceA := TE_602_MAVE_BLOCK.Out, SourceB := 60);
   TE_501_ROC := MUL_01.Dest;
   TE_504_ROC := MUL_02.Dest;
   TE_601_ROC := MUL_03.Dest;
   TE_602_ROC := MUL_04.Dest;
   SHEET 2
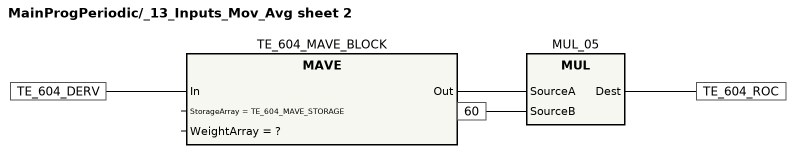
   TE_604_MAVE_BLOCK : MAVE(In := TE_604_DERV, StorageArray := TE_604_MAVE_STORAGE, WeightArray := ?);
   MUL_05 : MUL(SourceA := TE_604_MAVE_BLOCK.Out, SourceB := 60);
   TE_604_ROC := MUL_05.Dest;
END_ROUTINE

ROUTINE _13_Inputs_Rates   (* function block diagram *)
   SHEET 1
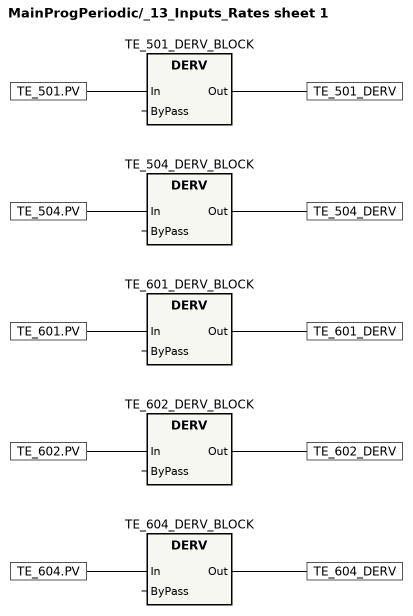
   TE_501_DERV_BLOCK : DERV(In := TE_501.PV);   // unwired pins: ByPass
   TE_504_DERV_BLOCK : DERV(In := TE_504.PV);   // unwired pins: ByPass
   TE_601_DERV_BLOCK : DERV(In := TE_601.PV);   // unwired pins: ByPass
   TE_602_DERV_BLOCK : DERV(In := TE_602.PV);   // unwired pins: ByPass
   TE_604_DERV_BLOCK : DERV(In := TE_604.PV);   // unwired pins: ByPass
   TE_501_DERV := TE_501_DERV_BLOCK.Out;
   TE_504_DERV := TE_504_DERV_BLOCK.Out;
   TE_601_DERV := TE_601_DERV_BLOCK.Out;
   TE_602_DERV := TE_602_DERV_BLOCK.Out;
   TE_604_DERV := TE_604_DERV_BLOCK.Out;
END_ROUTINE

ROUTINE _45_Process_PID_Control   (* function block diagram *)
// PID Control Blocks
   SHEET 1   // PIDE_101A
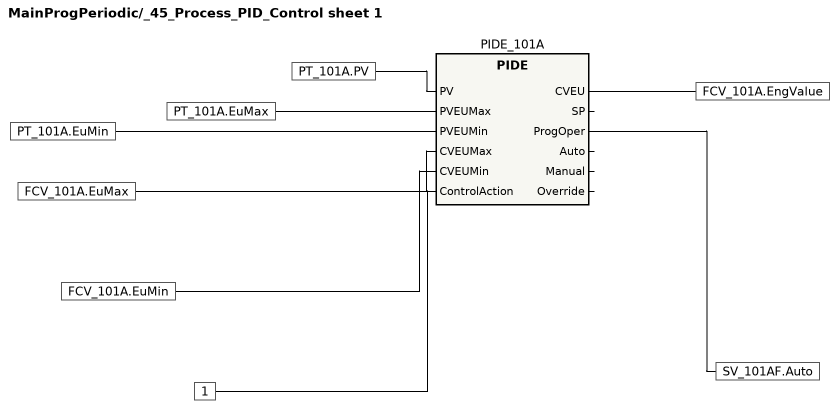
   PIDE_101A : PIDE(PV := PT_101A.PV, PVEUMax := PT_101A.EuMax, PVEUMin := PT_101A.EuMin, CVEUMax := FCV_101A.EuMax, CVEUMin := FCV_101A.EuMin, ControlAction := 1);   // unwired pins: SP Auto Manual Override
   FCV_101A.EngValue := PIDE_101A.CVEU;
   SV_101AF.Auto := PIDE_101A.ProgOper;
   SHEET 2   // PIDE_101B
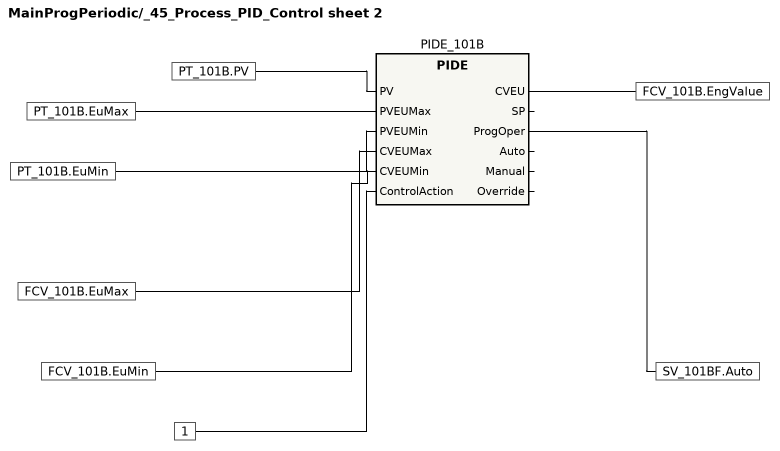
   PIDE_101B : PIDE(PV := PT_101B.PV, PVEUMax := PT_101B.EuMax, PVEUMin := PT_101B.EuMin, CVEUMax := FCV_101B.EuMax, CVEUMin := FCV_101B.EuMin, ControlAction := 1);   // unwired pins: SP Auto Manual Override
   FCV_101B.EngValue := PIDE_101B.CVEU;
   SV_101BF.Auto := PIDE_101B.ProgOper;
   SHEET 3   // PIDE_101C
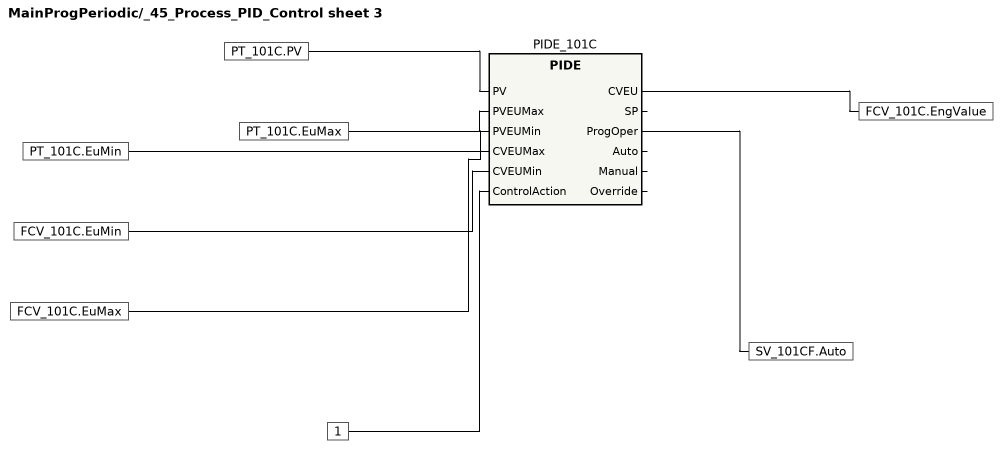
   PIDE_101C : PIDE(PV := PT_101C.PV, PVEUMax := PT_101C.EuMax, PVEUMin := PT_101C.EuMin, CVEUMax := FCV_101C.EuMax, CVEUMin := FCV_101C.EuMin, ControlAction := 1);   // unwired pins: SP Auto Manual Override
   SV_101CF.Auto := PIDE_101C.ProgOper;
   FCV_101C.EngValue := PIDE_101C.CVEU;
   SHEET 4   // PIDE_102A
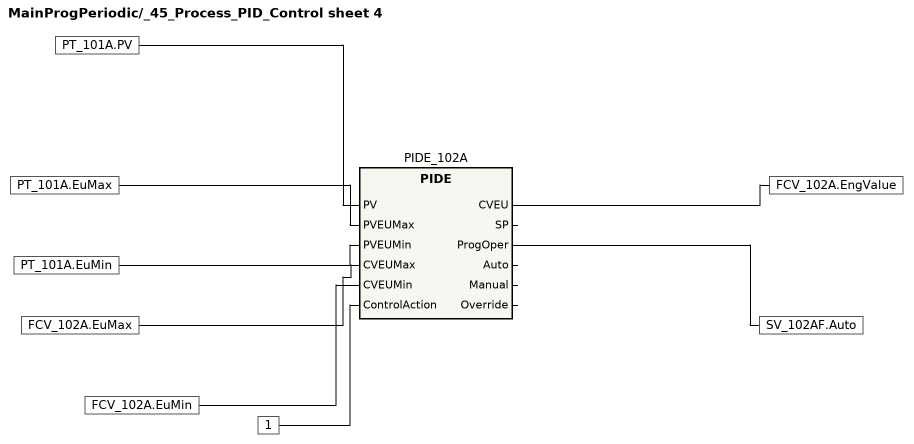
   PIDE_102A : PIDE(PV := PT_101A.PV, PVEUMax := PT_101A.EuMax, PVEUMin := PT_101A.EuMin, CVEUMax := FCV_102A.EuMax, CVEUMin := FCV_102A.EuMin, ControlAction := 1);   // unwired pins: SP Auto Manual Override
   SV_102AF.Auto := PIDE_102A.ProgOper;
   FCV_102A.EngValue := PIDE_102A.CVEU;
   SHEET 5   // PIDE_102B
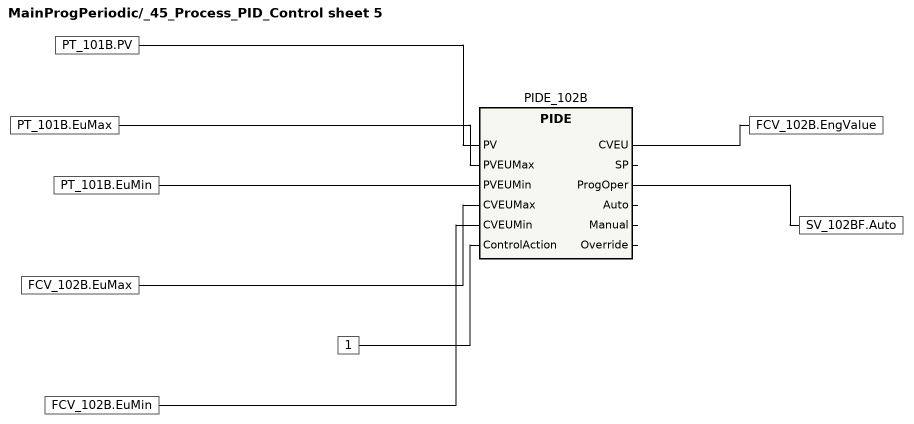
   PIDE_102B : PIDE(PV := PT_101B.PV, PVEUMax := PT_101B.EuMax, PVEUMin := PT_101B.EuMin, CVEUMax := FCV_102B.EuMax, CVEUMin := FCV_102B.EuMin, ControlAction := 1);   // unwired pins: SP Auto Manual Override
   FCV_102B.EngValue := PIDE_102B.CVEU;
   SV_102BF.Auto := PIDE_102B.ProgOper;
   SHEET 6   // PIDE_102C
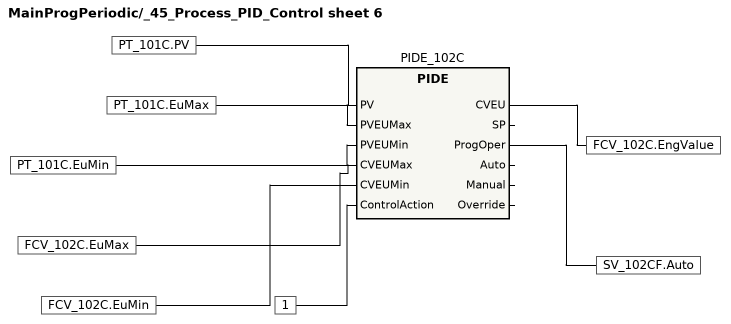
   PIDE_102C : PIDE(PV := PT_101C.PV, PVEUMax := PT_101C.EuMax, PVEUMin := PT_101C.EuMin, CVEUMax := FCV_102C.EuMax, CVEUMin := FCV_102C.EuMin, ControlAction := 1);   // unwired pins: SP Auto Manual Override
   FCV_102C.EngValue := PIDE_102C.CVEU;
   SV_102CF.Auto := PIDE_102C.ProgOper;
   SHEET 7   // PIDE_202
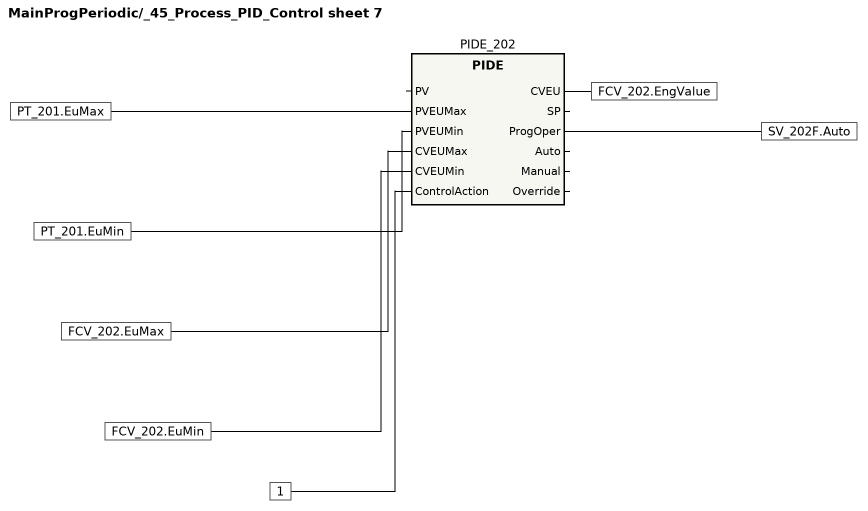
   PIDE_202 : PIDE(PVEUMax := PT_201.EuMax, PVEUMin := PT_201.EuMin, CVEUMax := FCV_202.EuMax, CVEUMin := FCV_202.EuMin, ControlAction := 1);   // unwired pins: PV SP Auto Manual Override
   FCV_202.EngValue := PIDE_202.CVEU;
   SV_202F.Auto := PIDE_202.ProgOper;
   SHEET 8   // PIDE_204
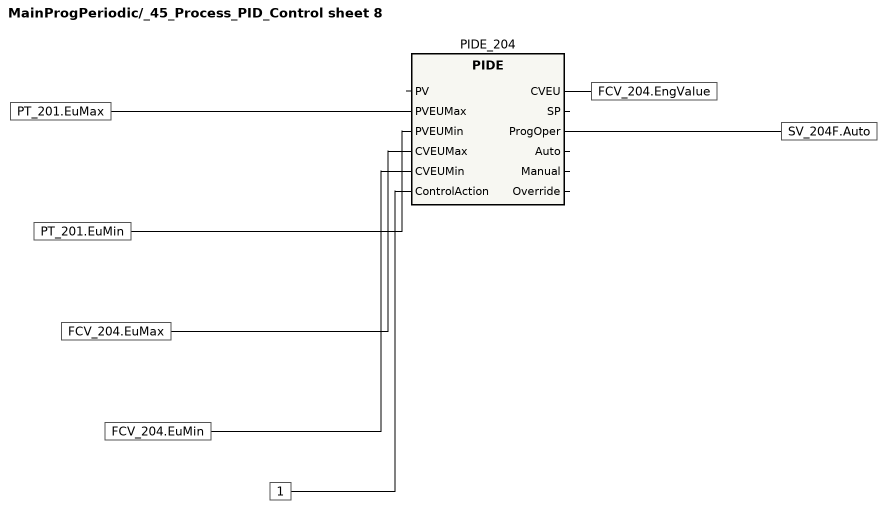
   PIDE_204 : PIDE(PVEUMax := PT_201.EuMax, PVEUMin := PT_201.EuMin, CVEUMax := FCV_204.EuMax, CVEUMin := FCV_204.EuMin, ControlAction := 1);   // unwired pins: PV SP Auto Manual Override
   FCV_204.EngValue := PIDE_204.CVEU;
   SV_204F.Auto := PIDE_204.ProgOper;
   SHEET 9   // PIDE_207
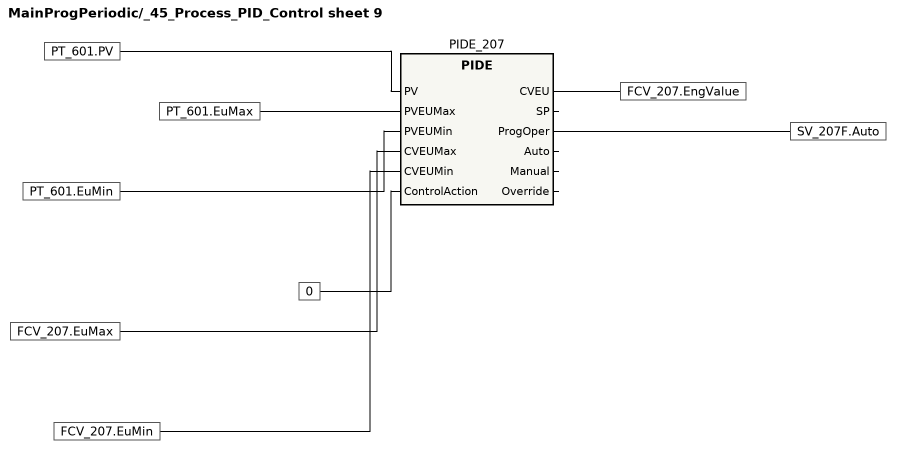
   PIDE_207 : PIDE(PV := PT_601.PV, PVEUMax := PT_601.EuMax, PVEUMin := PT_601.EuMin, CVEUMax := FCV_207.EuMax, CVEUMin := FCV_207.EuMin, ControlAction := 0);   // unwired pins: SP Auto Manual Override
   FCV_207.EngValue := PIDE_207.CVEU;
   SV_207F.Auto := PIDE_207.ProgOper;
   SHEET 10   // PIDE_504
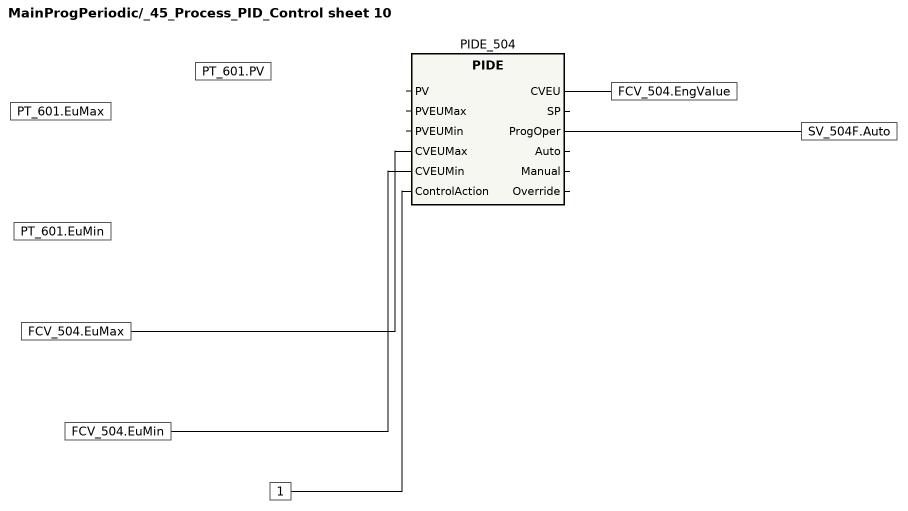
   // unwired input reference PT_601.EuMax
   // unwired input reference PT_601.EuMin
   // unwired input reference PT_601.PV
   PIDE_504 : PIDE(CVEUMax := FCV_504.EuMax, CVEUMin := FCV_504.EuMin, ControlAction := 1);   // unwired pins: PV PVEUMax PVEUMin SP Auto Manual Override
   FCV_504.EngValue := PIDE_504.CVEU;
   SV_504F.Auto := PIDE_504.ProgOper;
   SHEET 11   // PIDE_603
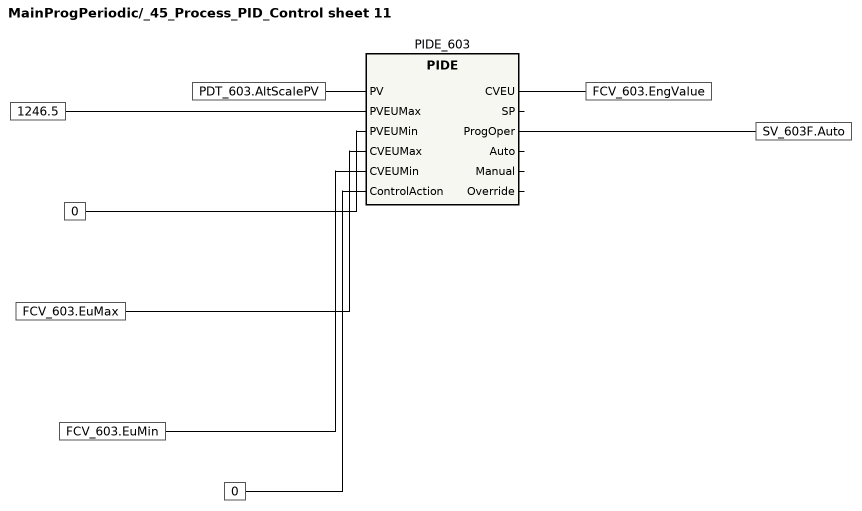
   PIDE_603 : PIDE(PV := PDT_603.AltScalePV, PVEUMax := 1246.5, PVEUMin := 0, CVEUMax := FCV_603.EuMax, CVEUMin := FCV_603.EuMin, ControlAction := 0);   // unwired pins: SP Auto Manual Override
   FCV_603.EngValue := PIDE_603.CVEU;
   SV_603F.Auto := PIDE_603.ProgOper;
   SHEET 12   // PIDE_605
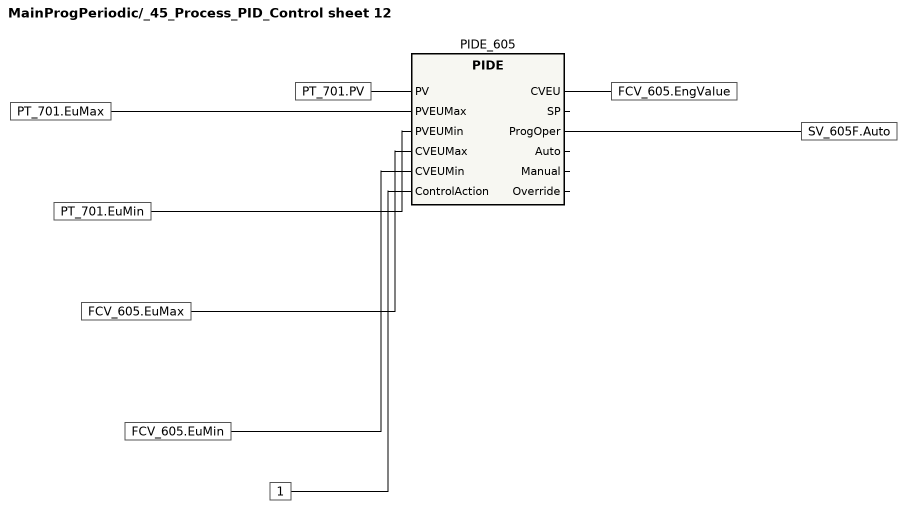
   PIDE_605 : PIDE(PV := PT_701.PV, PVEUMax := PT_701.EuMax, PVEUMin := PT_701.EuMin, CVEUMax := FCV_605.EuMax, CVEUMin := FCV_605.EuMin, ControlAction := 1);   // unwired pins: SP Auto Manual Override
   FCV_605.EngValue := PIDE_605.CVEU;
   SV_605F.Auto := PIDE_605.ProgOper;
   SHEET 13   // PIDE_753
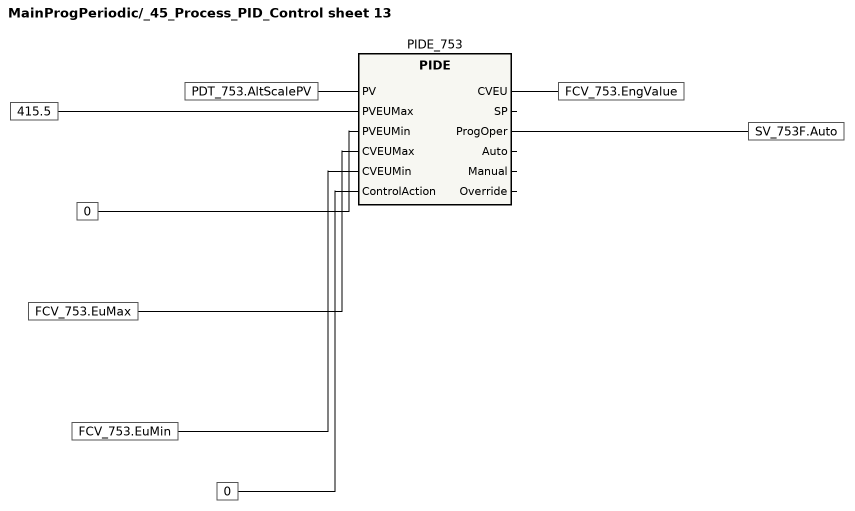
   PIDE_753 : PIDE(PV := PDT_753.AltScalePV, PVEUMax := 415.5, PVEUMin := 0, CVEUMax := FCV_753.EuMax, CVEUMin := FCV_753.EuMin, ControlAction := 0);   // unwired pins: SP Auto Manual Override
   FCV_753.EngValue := PIDE_753.CVEU;
   SV_753F.Auto := PIDE_753.ProgOper;
   SHEET 14   // PIDE_754
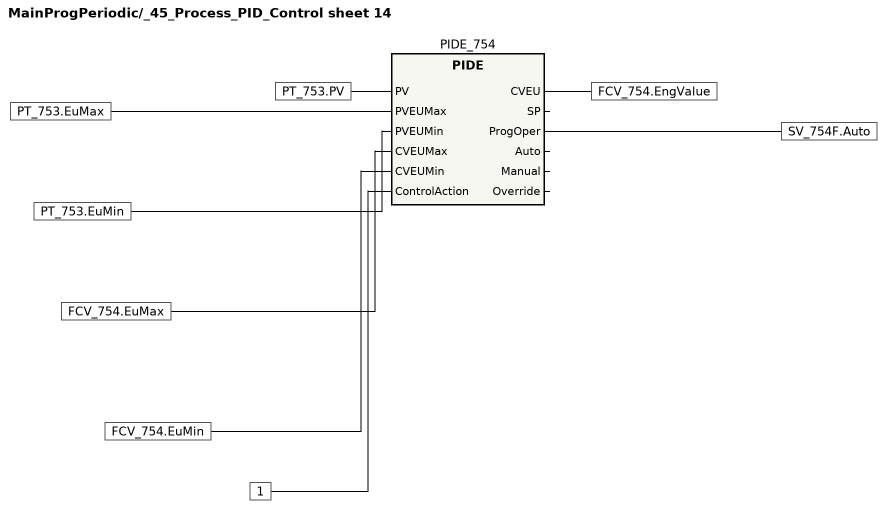
   PIDE_754 : PIDE(PV := PT_753.PV, PVEUMax := PT_753.EuMax, PVEUMin := PT_753.EuMin, CVEUMax := FCV_754.EuMax, CVEUMin := FCV_754.EuMin, ControlAction := 1);   // unwired pins: SP Auto Manual Override
   FCV_754.EngValue := PIDE_754.CVEU;
   SV_754F.Auto := PIDE_754.ProgOper;
   SHEET 15   // PIDE_755
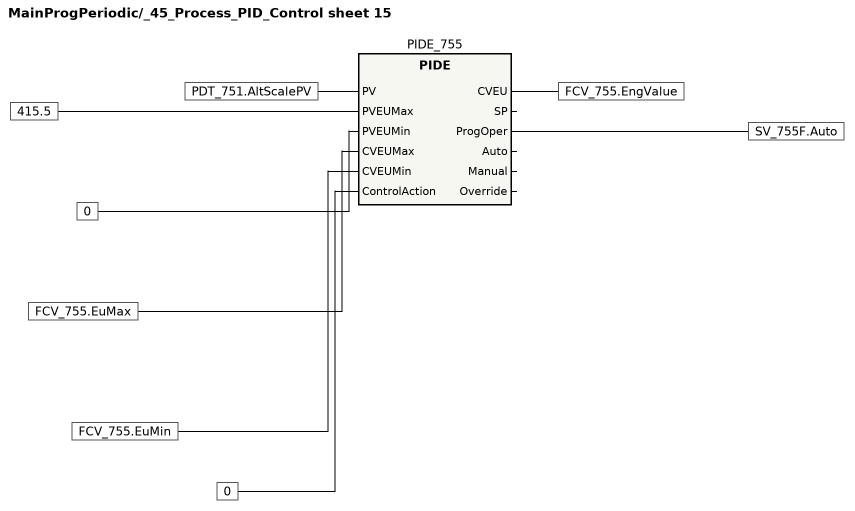
   PIDE_755 : PIDE(PV := PDT_751.AltScalePV, PVEUMax := 415.5, PVEUMin := 0, CVEUMax := FCV_755.EuMax, CVEUMin := FCV_755.EuMin, ControlAction := 0);   // unwired pins: SP Auto Manual Override
   FCV_755.EngValue := PIDE_755.CVEU;
   SV_755F.Auto := PIDE_755.ProgOper;
   SHEET 16   // PIDE_800
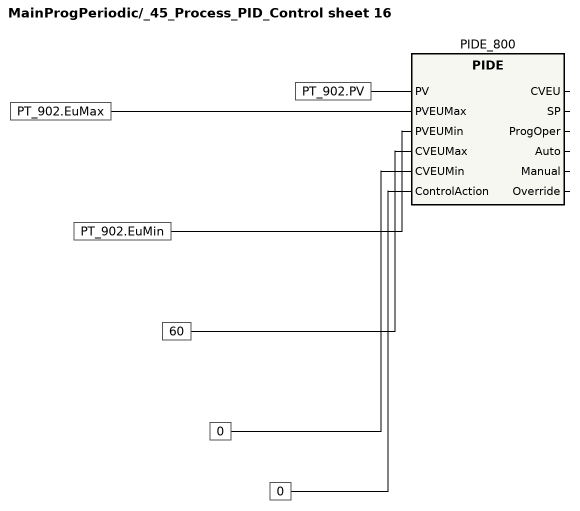
   PIDE_800 : PIDE(PV := PT_902.PV, PVEUMax := PT_902.EuMax, PVEUMin := PT_902.EuMin, CVEUMax := 60, CVEUMin := 0, ControlAction := 0);   // unwired pins: CVEU SP ProgOper Auto Manual Override
   SHEET 17   // PIDE_1001
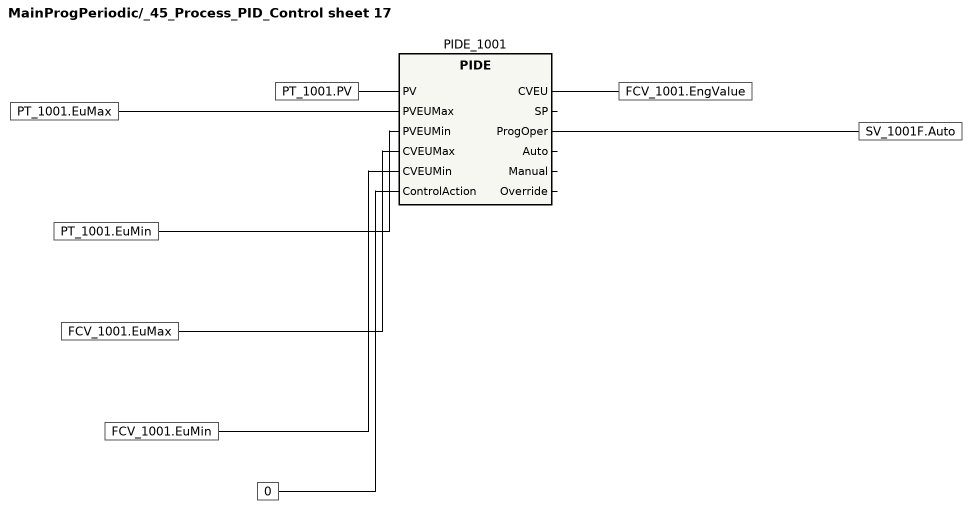
   PIDE_1001 : PIDE(PV := PT_1001.PV, PVEUMax := PT_1001.EuMax, PVEUMin := PT_1001.EuMin, CVEUMax := FCV_1001.EuMax, CVEUMin := FCV_1001.EuMin, ControlAction := 0);   // unwired pins: SP Auto Manual Override
   FCV_1001.EngValue := PIDE_1001.CVEU;
   SV_1001F.Auto := PIDE_1001.ProgOper;
   SHEET 18   // PIDE_1002
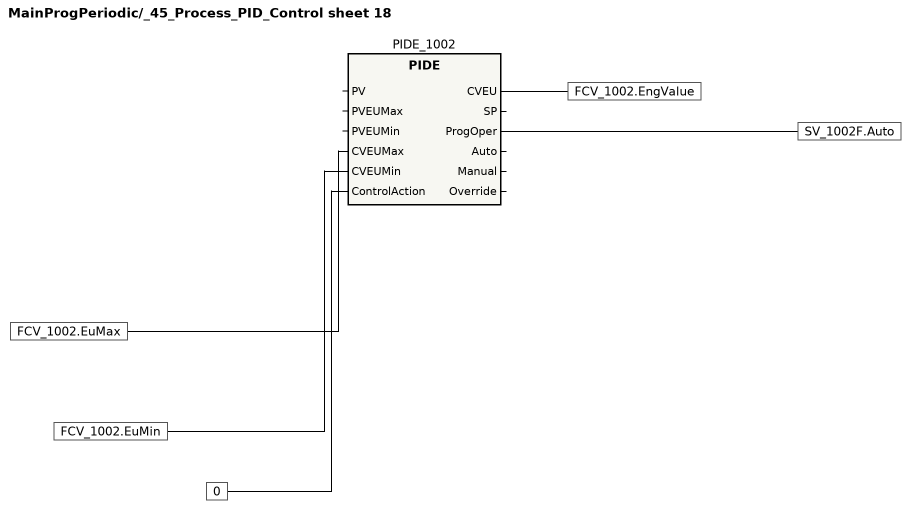
   PIDE_1002 : PIDE(CVEUMax := FCV_1002.EuMax, CVEUMin := FCV_1002.EuMin, ControlAction := 0);   // unwired pins: PV PVEUMax PVEUMin SP Auto Manual Override
   FCV_1002.EngValue := PIDE_1002.CVEU;
   SV_1002F.Auto := PIDE_1002.ProgOper;
   SHEET 19   // PIDE_1221
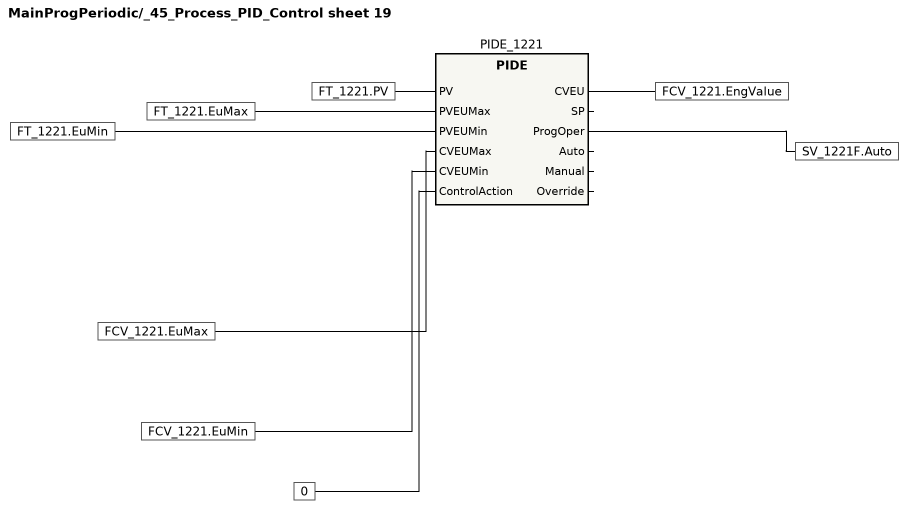
   PIDE_1221 : PIDE(PV := FT_1221.PV, PVEUMax := FT_1221.EuMax, PVEUMin := FT_1221.EuMin, CVEUMax := FCV_1221.EuMax, CVEUMin := FCV_1221.EuMin, ControlAction := 0);   // unwired pins: SP Auto Manual Override
   FCV_1221.EngValue := PIDE_1221.CVEU;
   SV_1221F.Auto := PIDE_1221.ProgOper;
   SHEET 20   // PIDE_1251
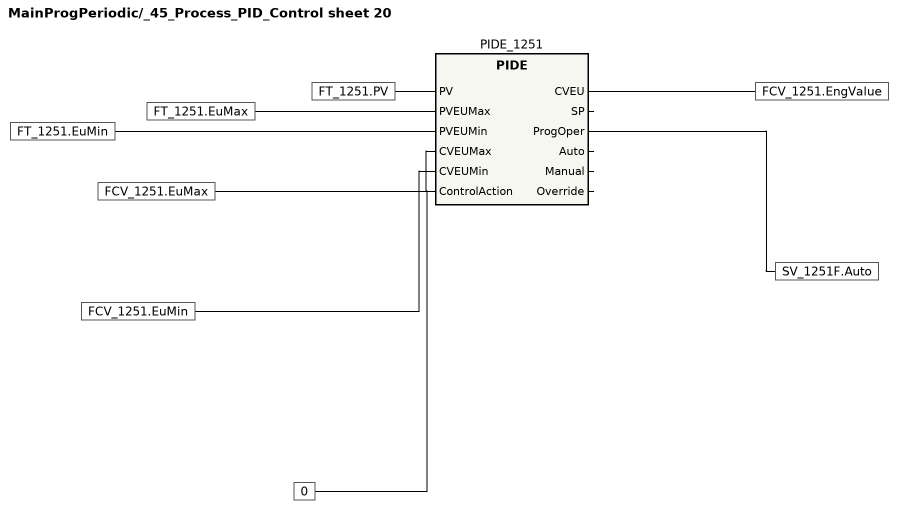
   PIDE_1251 : PIDE(PV := FT_1251.PV, PVEUMax := FT_1251.EuMax, PVEUMin := FT_1251.EuMin, CVEUMax := FCV_1251.EuMax, CVEUMin := FCV_1251.EuMin, ControlAction := 0);   // unwired pins: SP Auto Manual Override
   FCV_1251.EngValue := PIDE_1251.CVEU;
   SV_1251F.Auto := PIDE_1251.ProgOper;
END_ROUTINE
